Universal Robots PolyScope program: DoneRoboProg2.urp

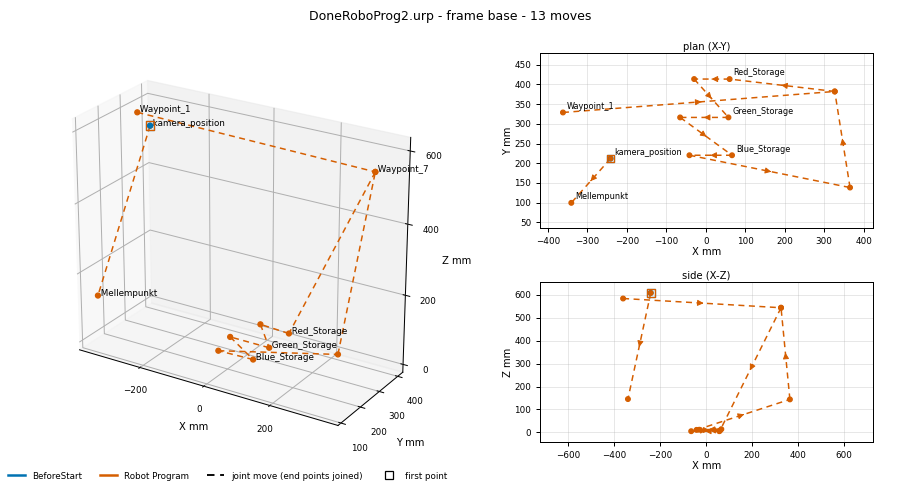
[picture p0: tool path of DoneRoboProg2.urp in frame base, 13 of 14 moves have a stored position in this frame; points joined in program order, loops and branches not executed]
Program DoneRoboProg2 (installation=default directory=/programs/usbdisk_1/RoboCop createdIn=3.9.1.64192 lastSavedIn=3.9.1.64192 robotSerialNumber=2016331617)
Calibrated DH parameters: a=[-0.000045, -0.22956, -0.153032, 0.000019, 0.0001, 0]; d=[0.152163, -856.35044, 904.692211, -48.229373, 0.085425, 0.082565]; alpha=[1.571202, -0.000097, 0.003084, 1.571016, -1.571253, 0]; deltaTheta=[-0.00003, 0.346154, 0.426056, -0.772366, 0.00006, 0.000029]
BeforeStart
  SuppressedNode
    Loop Counting (count=2) loopVariable(name=Loop_2)
      MoveJ speed 60 deg/s, acceleration 80 deg/s^2 (useActiveTCP=true)
        Waypoint Waypoint_2: TCP in base x=-436.649 y=121.636 z=16.057 mm, rx=-2.1976 ry=-2.2227 rz=-0.0328 rad; joints [-28.929, -55.196, 57.779, -93.137, -91.268, -0.822] deg; flange x=-437.533 y=115.27 z=260.973 mm, rx=-2.6752 ry=-1.6075 rz=-0.0257 rad
        Wait Sleep waitTime=1
        Waypoint Waypoint_4: TCP in base x=-220.9 y=121.569 z=16.045 mm, rx=-2.1975 ry=-2.2229 rz=-0.0327 rad; joints [-53.908, -107.202, 118.867, -102.756, -90.923, -25.791] deg; flange x=-221.776 y=115.235 z=260.962 mm, rx=-2.6752 ry=-1.6078 rz=-0.0256 rad
        Wait Sleep waitTime=1
        Waypoint Waypoint_5: TCP in base x=-220.86 y=276.516 z=16.029 mm, rx=-2.1977 ry=-2.2228 rz=-0.0327 rad; joints [-69.277, -81.318, 95.325, -105.335, -90.611, -41.146] deg; flange x=-221.742 y=270.18 z=260.946 mm, rx=-2.6753 ry=-1.6076 rz=-0.0256 rad
        Wait Sleep waitTime=1
  Script: Blue≟0
  Script: Green≟0
  Script: Red≟0
  Loop Forever
    Script: conres = socket_open("192.168.137.1",23)
    Script: textmsg(conres)
    If conres ≟  True
      Script: break
  Script: targetPos=p[0, 0, 0, 0, 0, 0]
  Script: receiveFromServ=[0, 0, 0, 0, 0, 0, 0, 0]
  MoveJ speed 60 deg/s, acceleration 80 deg/s^2 (useActiveTCP=true)
    Waypoint kamera_position: motionParameters(jointSpeed=1.047198 jointAcceleration=1.396263 cartesianSpeed=0.25 cartesianAcceleration=1.2); TCP in base x=-241.339 y=211.945 z=608.173 mm, rx=-1.5638 ry=0.0126 rz=-0.0738 rad; joints [0.457, -66.619, 23.973, -133.103, -183.621, 30.648] deg; flange x=-254.789 y=-32.679 z=606.358 mm, rx=-1.5202 ry=0.4013 rz=0.3196 rad
  Script: Kalibrer="Kalibrering"
  Script: socket_send_string(Kalibrer)
  Loop While (checkContinuously=false) expression=conres≟ True
    Script: KaliSlut=socket_read_ascii_float(1)
    Script: textmsg(KaliSlut)
    If KaliSlut[1]≟100
      Script: break
Robot Program (runOnlyOnce=false)
  Set DigitalOutput pin=tool_out[0]; digitalValue=0
  MoveJ speed 60 deg/s, acceleration 80 deg/s^2 (useActiveTCP=true)
    Waypoint kamera_position: TCP in base x=-241.339 y=211.945 z=608.173 mm, rx=-1.5638 ry=0.0126 rz=-0.0738 rad; joints [0.457, -66.619, 23.973, -133.103, -183.621, 30.648] deg; flange x=-254.789 y=-32.679 z=606.358 mm, rx=-1.5202 ry=0.4013 rz=0.3196 rad
  Wait Sleep waitTime=1.2
  Script: sendToServer="Klar"
  Script: socket_send_string(sendToServer)
  Wait Sleep waitTime=0.5
  Script: Modtaget = "Koordinater modtaget"
  SuppressedNode
    Script: socket_send_string(Modtaget)
  Loop While (checkContinuously=false) expression=conres≟ True
    Script: receiveFromServ=socket_read_ascii_float(7)
    Script: textmsg(receiveFromServ)
    If receiveFromServ[7]≟1
      Script: break
    ElseIf receiveFromServ[7]≟2
      Script: break
    ElseIf receiveFromServ[7]≟3
      Script: break
    ElseIf receiveFromServ[7]≟4
      Script: break
  Loop Forever
    MoveJ speed 60 deg/s, acceleration 80 deg/s^2 (useActiveTCP=true)
      Waypoint Mellempunkt: TCP in base x=-340.682 y=99.742 z=145.518 mm, rx=3.0999 ry=-0.0003 rz=0.0001 rad; joints [-36.703, -75.687, 51.77, -64.672, -87.906, 81.977] deg; flange x=-340.702 y=109.942 z=390.306 mm, rx=3.0047 ry=-0.7675 rz=0.0161 rad
    Script: targetPos=p[receiveFromServ[1],receiveFromServ[2],receiveFromServ[3],receiveFromServ[4],receiveFromServ[5],receiveFromServ[6]]
    Script: textmsg(targetPos)
    If targetPos≠p[0, 0, 0, 0, 0, 0]
      MoveJ speed 60 deg/s, acceleration 80 deg/s^2 (useActiveTCP=true)
        Waypoint Waypoint (Variable): variable=targetPos
      Script: break
  Set ExpressionOutput pin=tool_out[0]; expression=True
  Wait DigitalInput pin=tool_in[0]; digitalValue=1
  MoveJ speed 60 deg/s, acceleration 80 deg/s^2 (useActiveTCP=true)
    Waypoint Waypoint_1: TCP in base x=-361.802 y=328.652 z=583.927 mm, rx=-1.5551 ry=-0.7269 rz=0.4118 rad; joints [-70.552, -98.81, 54.815, -128.179, -68.723, 16.754] deg; flange x=-202.745 y=144.977 z=615.378 mm, rx=-1.7317 ry=-0.3281 rz=0.7783 rad
    Waypoint Waypoint_7: TCP in base x=326.746 y=381.88 z=543.632 mm, rx=-1.7283 ry=0.6111 rz=-0.6667 rad; joints [-157.994, -98.304, 58.726, -127.451, -68.738, 16.754] deg; flange x=153.756 y=216.243 z=595.242 mm, rx=-1.4906 ry=0.9978 rz=-0.3122 rad
  Wait Sleep waitTime=2
  If receiveFromServ[7]≟1
    If Red≟0
      MoveJ speed 60 deg/s, acceleration 80 deg/s^2 (useActiveTCP=true)
        Waypoint Red_Storage: TCP in base x=60.403 y=413.236 z=7.687 mm, rx=3.1337 ry=-0.0907 rz=0.0118 rad; joints [-113.548, -63.697, 73.189, -99.319, -90.418, 8.545] deg; flange x=58.613 y=414.899 z=252.675 mm, rx=3.0158 ry=-0.8637 rz=0.0139 rad
        Set ExpressionOutput pin=tool_out[0]; expression=False
        Wait Sleep waitTime=1
        Set IncrementVariable installationVariable=Red
    ElseIf Red≠0
      MoveJ speed 60 deg/s, acceleration 80 deg/s^2 (useActiveTCP=true)
        Waypoint Red_Storage_2: TCP in base x=-29.487 y=413.323 z=11.81 mm, rx=-3.1349 ry=0.0177 rz=-0.0013 rad; joints [-101.74, -65.647, 75.215, -99.969, -89.852, 17.686] deg; flange x=-29.702 y=411.69 z=256.804 mm, rx=-3.033 ry=0.7927 rz=0.0013 rad
        Set ExpressionOutput pin=tool_out[0]; expression=False
        Wait Sleep waitTime=1
  ElseIf receiveFromServ[7]≟2
    If Green≟0
      MoveJ speed 60 deg/s, acceleration 80 deg/s^2 (useActiveTCP=true)
        Waypoint Green_Storage: TCP in base x=57.429 y=316.13 z=5.393 mm, rx=-3.1399 ry=0.0479 rz=-0.0041 rad; joints [-120.752, -87.426, 104.591, -107.322, -89.992, -0.212] deg; flange x=56.779 y=315.82 z=250.392 mm, rx=-3.0299 ry=0.8231 rz=-0.0035 rad
        Set ExpressionOutput pin=tool_out[0]; expression=False
        Wait Sleep waitTime=1
        Set IncrementVariable installationVariable=Green
    ElseIf Green≠0
      MoveJ speed 60 deg/s, acceleration 80 deg/s^2 (useActiveTCP=true)
        Waypoint Green_Storage_2: TCP in base x=-64.938 y=316.074 z=5.367 mm, rx=3.1213 ry=0 rz=0.0001 rad; joints [-98.664, -85.473, 101.98, -105.378, -90.071, 20.128] deg; flange x=-64.951 y=321.036 z=250.317 mm, rx=3.0249 ry=-0.7724 rz=0.0079 rad
        Set ExpressionOutput pin=tool_out[0]; expression=False
        Wait Sleep waitTime=1
  ElseIf receiveFromServ[7]≟3
    If Blue≟0
      MoveJ speed 60 deg/s, acceleration 80 deg/s^2 (useActiveTCP=true)
        Waypoint Blue_Storage: TCP in base x=66.483 y=220.275 z=14.072 mm, rx=3.134 ry=0.0002 rz=0.0001 rad; joints [-135.646, -112.288, 121.903, -99.328, -90.188, -16.874] deg; flange x=66.472 y=222.137 z=259.065 mm, rx=3.0369 ry=-0.7752 rz=0.003 rad
        Set ExpressionOutput pin=tool_out[0]; expression=False
        Wait Sleep waitTime=1
        Set IncrementVariable installationVariable=Blue
    ElseIf Blue≠0
      MoveJ speed 60 deg/s, acceleration 80 deg/s^2 (useActiveTCP=true)
        Waypoint Blue_Storage_2: TCP in base x=-41.402 y=220.28 z=11.151 mm, rx=3.1237 ry=-0.0002 rz=0.0003 rad; joints [-108.994, -112.995, 122.832, -98.888, -90.218, 9.793] deg; flange x=-41.451 y=224.665 z=256.112 mm, rx=3.0271 ry=-0.7731 rz=0.0072 rad
        Set ExpressionOutput pin=tool_out[0]; expression=False
        Wait Sleep waitTime=1
  ElseIf receiveFromServ[7]≟4
    MoveJ speed 60 deg/s, acceleration 80 deg/s^2 (useActiveTCP=true)
      Waypoint Skrald: TCP in base x=365.434 y=138.467 z=144.008 mm, rx=-2.8359 ry=-1.1412 rz=-0.3218 rad; joints [-183.779, -86.964, 72.213, -84.491, -81.164, -108.165] deg; flange x=324.323 y=104.122 z=383.08 mm, rx=-2.9845 ry=-0.3981 rz=-0.2817 rad
      Set ExpressionOutput pin=tool_out[0]; expression=False
      Wait Sleep waitTime=1
  Wait Sleep waitTime=1
  Script: targetPos=p[0, 0, 0, 0, 0, 0]
  MoveJ speed 60 deg/s, acceleration 80 deg/s^2 (useActiveTCP=true)
    Waypoint Waypoint_7: TCP in base x=326.746 y=381.88 z=543.632 mm, rx=-1.7283 ry=0.6111 rz=-0.6667 rad; joints [-157.994, -98.304, 58.726, -127.451, -68.738, 16.754] deg; flange x=153.756 y=216.243 z=595.242 mm, rx=-1.4906 ry=0.9978 rz=-0.3122 rad
